DATA_BLOCK "FB_ParameterTypes_DB"
{ S7_Optimized_Access := 'TRUE' }
VERSION : 0.1
NON_RETAIN
"FB_ParameterTypes"

BEGIN

END_DATA_BLOCK

